FUNCTION_BLOCK Msg3001_HoldRelease EXTENDS TcpIpCommandResultFilter IMPLEMENTS I_Navitrol_ReturnToRoute
VAR
	Command		  : ST_TcpIpPayload;
	ReceiveBuffer : U_Recived_bytes_from_Navitrol;
	ReleaseHold	  : ST_3001_ReleaseHoldState;
	HoldReleased  : ST_3101_HoldReleased;
END_VAR

METHOD Execute : BOOL
IF TcpIpConnection.ConnectionState = eSOCKET_CONNECTED THEN
	F_SetHeaderInfo(ReleaseHold);
	MEMSET(ADR(Command), 0, SIZEOF(Command));
	Command.Size := SIZEOF(ReleaseHold);
	MEMCPY(ADR(Command.Data), ADR(ReleaseHold), Command.Size);
	TcpIpConnection.SendCommand(ADR(Command));
	CommandActive := TRUE;
	Execute		  := TRUE;
END_IF
END_METHOD

METHOD UpdateCommandResult
VAR_INPUT
	Response : POINTER TO ST_TcpIpPayload;
END_VAR

VAR_INST
	ReceiveCounter : UDINT;
END_VAR
MEMCPY(ADR(ReceiveBuffer), ADR(Response^.Data), SIZEOF(ReceiveBuffer));
IF ReceiveBuffer.Header.Message_ID = 3101 THEN
	ReceiveCounter := ReceiveCounter + 1;
	MEMCPY(destAddr := ADR(HoldReleased), srcAddr := ADR(ReceiveBuffer), n := SIZEOF(HoldReleased));
	CommandActive := FALSE;
END_IF
END_METHOD

END_FUNCTION_BLOCK

(* stored: Version 1.1.0.1
   POU Msg3001_HoldRelease: Id {6768bc0e-9991-49a4-8ec3-789fd55770e9}, SpecialFunc None
   Method Execute: Id {76f568aa-aa9b-40b0-9b99-e9742db5ad72}
   Method UpdateCommandResult: Id {6bcc92ca-0e66-4617-b04c-77d44c42869c} *)
